TYPE ST_MessageHeader :
STRUCT

	(*CreationDate 				: STRING(10);
	CreationTime 				: STRING(25);*)
	ReferenceID				: T_MaxString;
	CreationTimeLocalUTC		: T_ISO8601Time;
	MessageType	 			: STRING(25);
	SenderSystem				: STRING(5);
	ReceiverSystem			: STRING(5);


END_STRUCT
END_TYPE

(* stored: Version 1.1.0.1, ProductVersion 3.1.4024.15
   DUT ST_MessageHeader: Id {785d0490-46b4-4a7d-b08e-39e5edbd2045} *)
